// Mitsubishi GX Works2 project: 0715   PLC: Q02/Q02H

PROGRAM MAIN
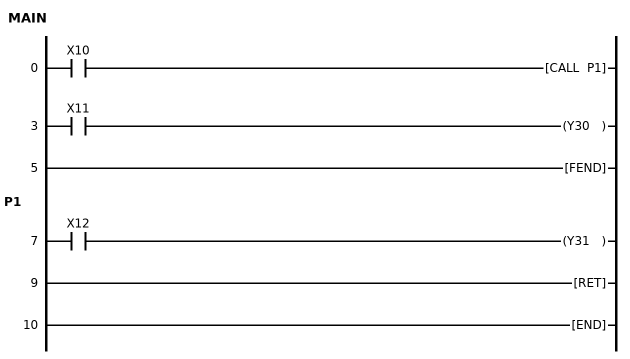
0     LD      X10
      CALL    P1
3     LD      X11
      OUT     Y30
5     FEND
      P1
7     LD      X12
      OUT     Y31
9     RET
10    END
END_PROGRAM

PROGRAM MAIN1
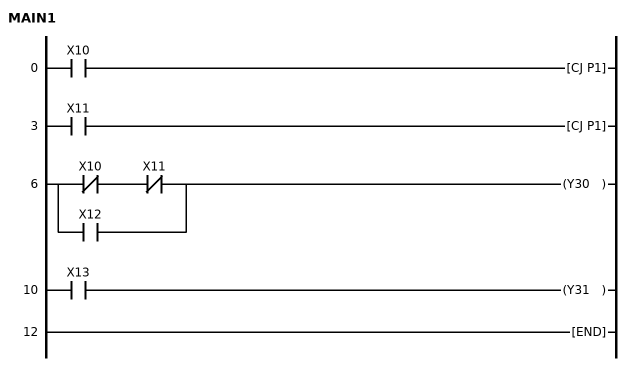
0     LD      X10
      CJ      P1
3     LD      X11
      SCJ     P1
6     LDI     X10
      ANI     X11
      OR      X12
      OUT     Y30
10    LD      X13
      OUT     Y31
12    END
END_PROGRAM

PROGRAM MAIN2
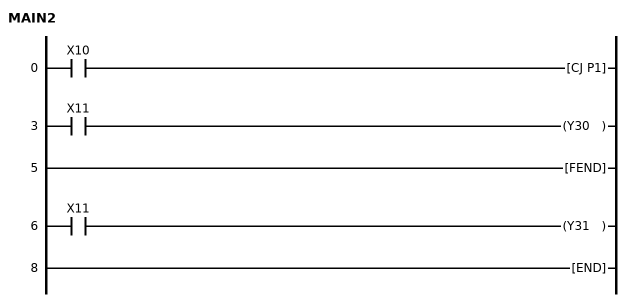
0     LD      X10
      CJ      P1
3     LD      X11
      OUT     Y30
5     FEND
6     LD      X11
      OUT     Y31
8     END
END_PROGRAM
